FUNCTION_BLOCK FbReset
TITLE = 'FbReset'
//Флаг первого скана с TOF задержкой выключен CFC PCS7.

{//FB attributes for PCS7.
S7_tasklist := 'OB100' //Call in OB100
}

VERSION : '1.0'
AUTHOR  : VA
FAMILY  : LIB_PLC

VAR_INPUT
TimeDelayOff
{//Атрибуты переменных PCS7.
S7_link    := 'false'; //'false' запрет CFC соединений.
S7_dynamic := 'true'   //'true' просмотр в CFC.
} : DINT := 1000; //Задержка выключен. импульса сброса ms.
END_VAR

VAR_OUTPUT
Reset :BOOL := FALSE; //Сброс алгоритма.
END_VAR

VAR
RST :BOOL := FALSE; //Сброс алгоритма локальный.
TOF1 : SFB5; //TOF timer.
END_VAR

VAR_TEMP
TOP_SI: STRUCT
    EV_CLASS :BYTE ;
    EV_NUM   :BYTE ;
    PRIORITY :BYTE ;
    NUM      :BYTE ;
    TYP2_3   :BYTE ;
    TYP1     :BYTE ;
    ZI1      :WORD ;
    ZI2_3    :DWORD;
END_STRUCT;
START_UP_SI: STRUCT
    EV_CLASS :BYTE ;
    EV_NUM   :BYTE ;
    PRIORITY :BYTE ;
    NUM      :BYTE ;
    TYP2_3   :BYTE ;
    TYP1     :BYTE ;
    ZI1      :WORD ;
    ZI2_3    :DWORD;
END_STRUCT;
ERROR_RD_SINFO :INT;
END_VAR

//Анализ из какого OB произошел вызов.
//Штатно вызов из OB35 или другой цикличный.
//При перезагрузке вызов из OB100.
ERROR_RD_SINFO := SFC6(TOP_SI := TOP_SI, START_UP_SI := START_UP_SI); //RD_SINFO
RST := (TOP_SI.NUM = 100); //Call in OB100

//Задержка выключен. импульса первого скана.
IF (TimeDelayOff <= 0) THEN
TOF1.IN := FALSE;
TOF1.PT := T#0ms;
TOF1();
Reset := RST;
ELSE
TOF1.IN := RST;
TOF1.PT := DINT_TO_TIME(TimeDelayOff);
TOF1();
Reset := TOF1.Q; // OUT: BOOL
END_IF;

END_FUNCTION_BLOCK

//Блок спроектирован под PCS7 v5.

//  +---------+
//  | GNU GPL |
//  +---------+
//  |
//  |
//  .= .-_-. =.
// ((_/)o o(\_))
//  `-'(. .)`-'
//  |/| \_/ |\
//  ( |     | )
//  /"\_____/"\
//  \__)   (__/
// @COPYLEFT ALL WRONGS RESERVED :)
// Author: VA
// Contacts: DIY.PLC.314@gmail.com
// License: GNU GPL v2
//
// https://www.youtube.com/@DIY_PLC
// https://github.com/DIYPLC
